// TwinCAT 3 PLC project PLC
// ProgramVersion: 3.1.4026.19
// CompilerDefines: VISU_USEPROPERTYINFO
// libraries:
//   SPT Base Types, * (Beckhoff Automation LLC)
//   SPT Components, * (Beckhoff Automation LLC)
//   SPT Motion Control, * (Beckhoff Automation LLC)
//   SPT Utilities, * (Beckhoff Automation LLC)
//   Tc2_Standard, * (Beckhoff Automation GmbH)
//   Tc2_System, * (Beckhoff Automation GmbH)
//   Tc3_PackML_V3, * (Beckhoff Automation GmbH)
// project tree:
//   DUTs/ E_PMLCustomMode.TcDUT, ST_ModeList.TcDUT
//   / GlobalTextList.TcGTLO, PlcTask.TcTTO, Visualization Manager.TcVMO (not stored)
//   Modes/ FB_CustomModes.TcPOU
//   Modules/00 Machine/DUTs/ ST_Machine_Command.TcDUT, ST_Machine_Config.TcDUT, ST_Machine_HMI.TcDUT, ST_Machine_Status.TcDUT
//   Modules/00 Machine/ Machine.TcPOU
//   Modules/01 Infeed/ Infeed.TcPOU
//   Modules/02 Process/ Process.TcPOU
//   Modules/03 Outfeed/ Outfeed.TcPOU
//   POUs/ MAIN.TcPOU
//   VISUs/ Visualization.TcVIS
// real-time tasks:
//   TASK PlcTask: cycle T#10ms, priority 20, ADS port 350
// motion (NC):
//   TASK NC-Task 1 SAF: cycle T#2ms, priority 4, ADS port 501
//   TASK NC-Task 1 SVB: cycle T#10ms, priority 8, ADS port 511
//   AXIS Axis 1 (id 1)
// variable links:
//   PLC/PLC Instance <-> NC-Task 1 SAF/Axes/Axis 1
//     PlcTask Inputs/MAIN.Machine.Infeed.Axis.BasicAxis._Axis.NcToPlc <-> Outputs/ToPlc
//     PlcTask Outputs/MAIN.Machine.Infeed.Axis.BasicAxis._Axis.PlcToNc <-> Inputs/FromPlc

CONFIGURATION PLC
    RESOURCE PLC ON TwinCAT3
        TASK PlcTask(INTERVAL := T#10ms, PRIORITY := 20);
        PROGRAM MAIN WITH PlcTask : MAIN;
    END_RESOURCE
END_CONFIGURATION

// ---- DUTs/E_PMLCustomMode.TcDUT
{attribute 'to_string'}
TYPE E_PMLCustomMode : (
		//Protected
		Invalid		:= 0,
		Production	:= 1,
		Maintenance := 2,
		Manual		:= 3,
		//User-Defined
		Home		  := 4,	 //User Mode 1
		PrePosition	  := 5,	 //User Mode 2
		PreProduction := 6,	 //User Mode 3
		SingleCycle	  := 7,	 //User Mode 4
		SingleStep	  := 8,	 //User Mode 5
		Setup		  := 9,	 //User Mode 6
		CleanInPlace  := 10, //User Mode 7
		DryCycle	  := 11, //User Mode 8
		Teach		  := 12, //User Mode 9
		Remote		  := 13, //User Mode 10
		Last		  := 14	 //User Mode 11

	//E_PMLUnitMode.ePMLUnitMode_UserMode28
	) DINT;
END_TYPE

// ---- DUTs/ST_ModeList.TcDUT
TYPE ST_ModeList :
	STRUCT
		// Protected
		Invalid		: BOOL;
		Production	: BOOL;
		Maintenance : BOOL;
		Manual		: BOOL;
		// User-Defined
		Home		  : BOOL;
		PrePosition	  : BOOL;
		PreProduction : BOOL;
		SingleCycle	  : BOOL;
		SingleStep	  : BOOL;
		Setup		  : BOOL;
		CleanInPlace  : BOOL;
		DryCycle	  : BOOL;
		Teach		  : BOOL;
		Remote		  : BOOL;
		Last		  : BOOL;
		// Unused
		UserMode12 : BOOL;
		UserMode13 : BOOL;
		UserMode14 : BOOL;
		UserMode15 : BOOL;
		UserMode16 : BOOL;
		UserMode17 : BOOL;
		UserMode18 : BOOL;
		UserMode19 : BOOL;
		UserMode20 : BOOL;
		UserMode21 : BOOL;
		UserMode22 : BOOL;
		UserMode23 : BOOL;
		UserMode24 : BOOL;
		UserMode25 : BOOL;
		UserMode26 : BOOL;
		UserMode27 : BOOL;
		UserMode28 : BOOL;
	END_STRUCT
END_TYPE

// ---- Modules/00 Machine/DUTs/ST_Machine_Command.TcDUT
TYPE ST_Machine_Command :
	STRUCT
		StartHoming : BOOL;
	END_STRUCT
END_TYPE

// ---- Modules/00 Machine/DUTs/ST_Machine_Config.TcDUT
TYPE ST_Machine_Config :
	STRUCT
	END_STRUCT
END_TYPE

// ---- Modules/00 Machine/DUTs/ST_Machine_HMI.TcDUT
TYPE ST_Machine_HMI :
	STRUCT
		Command : ST_Machine_Command;
		Config	: ST_Machine_Config;
		Status	: ST_Machine_Status;
	END_STRUCT
END_TYPE

// ---- Modules/00 Machine/DUTs/ST_Machine_Status.TcDUT
TYPE ST_Machine_Status :
	STRUCT
		HomeComplete  : BOOL;
		NeedsCleaning : BOOL;
		CleanComplete : BOOL;
	END_STRUCT
END_TYPE

// ---- POUs/MAIN.TcPOU
PROGRAM MAIN
VAR
	Machine : Machine := (Name := 'Machine');
END_VAR

(*All sample code provided by Beckhoff Automation LLC are for illustrative purposes only and are provided “as is” and without any warranties, express or implied. Actual implementations in applications will vary significantly. Beckhoff Automation LLC shall have no liability for, and does not waive any rights in relation to, any code samples that it provides or the use of such code samples for any purpose.*)

(*
	This sample demonstrates changing mode based on the status of the machine.
	Specifically on startup, the Machine Status for HomeComplete is FALSE.
	Therefore in Machine.Idle the mode is changed to Home.
	When the 'Start command is given the Machine can then Execute its Homing routine, Complete, and then return to Idle.
	Once back in Idle, the Machine status of HomeComplete will retunr the mode to Production.
*)
Machine.CyclicLogic();

END_PROGRAM

// ---- Modules/00 Machine/Machine.TcPOU
FUNCTION_BLOCK Machine EXTENDS FB_PackML_BaseModule
VAR
	Infeed	: Infeed  := (Name := 'Infeed');
	Process : Process := (Name := 'Process');
	Outfeed : Outfeed := (Name := 'Outfeed');

	//
	Machine_HMI		  : ST_Machine_HMI;
	CurrentCustomMode : E_PMLCustomMode;
END_VAR

METHOD CreateCustomModes
VAR
	i		   : E_PMLCustomMode;
	aModeNames : ARRAY[E_PMLCustomMode.Invalid..E_PMLCustomMode.Last] OF STRING;
END_VAR
aModeNames[0]  := TO_STRING(E_PMLCustomMode.Invalid);
aModeNames[1]  := TO_STRING(E_PMLCustomMode.Production);
aModeNames[2]  := TO_STRING(E_PMLCustomMode.Maintenance);
aModeNames[3]  := TO_STRING(E_PMLCustomMode.Manual);
aModeNames[4]  := TO_STRING(E_PMLCustomMode.Home);			//UserMode1
aModeNames[5]  := TO_STRING(E_PMLCustomMode.PrePosition);	//UserMode2
aModeNames[6]  := TO_STRING(E_PMLCustomMode.PreProduction); //UserMode3
aModeNames[7]  := TO_STRING(E_PMLCustomMode.SingleCycle);	//UserMode4
aModeNames[8]  := TO_STRING(E_PMLCustomMode.SingleStep);	//UserMode5
aModeNames[9]  := TO_STRING(E_PMLCustomMode.Setup);			//UserMode6
aModeNames[10] := TO_STRING(E_PMLCustomMode.CleanInPlace);	//UserMode7
aModeNames[11] := TO_STRING(E_PMLCustomMode.DryCycle);		//UserMode8
aModeNames[12] := TO_STRING(E_PMLCustomMode.Teach);			//UserMode9
aModeNames[13] := TO_STRING(E_PMLCustomMode.Remote);		//UserMode10
aModeNames[14] := TO_STRING(E_PMLCustomMode.Last);			//UserMode11

//Default Config for all modes, this is also the default config for Production Mode as defined by Pack ML
CustomModes.bDisableClearing			   := FALSE;
CustomModes.bDisableStarting			   := FALSE;
CustomModes.bDisableSuspended			   := FALSE;
CustomModes.bDisableStopping			   := FALSE;
CustomModes.bDisableAborting			   := FALSE;
CustomModes.bDisableHolding				   := FALSE;
CustomModes.bDisableHeld				   := FALSE;
CustomModes.bDisableUnholding			   := FALSE;
CustomModes.bDisableSuspending			   := FALSE;
CustomModes.bDisableUnsuspending		   := FALSE;
CustomModes.bDisableResetting			   := FALSE;
CustomModes.bDisableIdle				   := FALSE;
CustomModes.bDisableCompleting			   := FALSE;
CustomModes.bDisableComplete			   := FALSE;
CustomModes.bEnableUnitModeChangeStopped   := TRUE;
CustomModes.bEnableUnitModeChangeIdle	   := TRUE;
CustomModes.bEnableUnitModeChangeSuspended := TRUE;
CustomModes.bEnableUnitModeChangeExecute   := FALSE;
CustomModes.bEnableUnitModeChangeAborted   := TRUE;
CustomModes.bEnableUnitModeChangeHeld	   := TRUE;
CustomModes.bEnableUnitModeChangeComplete  := TRUE;

//
FOR i := E_PMLCustomMode.Invalid TO E_PMLCustomMode.Last DO
	CustomModes(emode := i, sName := aModeNames[i]);
END_FOR

// Production - Changes for Clean In Place Mode to move from Production.Execute to CleanInPlace.Execute
CustomModes(eMode := E_PMLCustomMode.Production, sName := 'Production', bEnableUnitModeChangeExecute := TRUE);

//Maintenance Mode default as defined by PackML
CustomModes(eMode						   := E_PMLCustomMode.Maintenance,
			sName						   := 'Maintenance',
			bDisableClearing			   := FALSE,
			bDisableStarting			   := FALSE,
			bDisableSuspended			   := TRUE,
			bDisableStopping			   := FALSE,
			bDisableAborting			   := FALSE,
			bDisableHolding				   := FALSE,
			bDisableHeld				   := FALSE,
			bDisableUnholding			   := FALSE,
			bDisableSuspending			   := TRUE,
			bDisableUnsuspending		   := TRUE,
			bDisableResetting			   := FALSE,
			bDisableIdle				   := FALSE,
			bDisableCompleting			   := TRUE,
			bDisableComplete			   := TRUE,
			bEnableUnitModeChangeStopped   := TRUE,
			bEnableUnitModeChangeIdle	   := TRUE,
			bEnableUnitModeChangeSuspended := FALSE,
			bEnableUnitModeChangeExecute   := FALSE,
			bEnableUnitModeChangeAborted   := TRUE,
			bEnableUnitModeChangeHeld	   := TRUE,
			bEnableUnitModeChangeComplete  := FALSE);

//Manual Mode default as defined by PackML
CustomModes(eMode						   := E_PMLCustomMode.Manual,
			sName						   := 'Manual',
			bDisableClearing			   := FALSE,
			bDisableStarting			   := FALSE,
			bDisableSuspended			   := TRUE,
			bDisableStopping			   := FALSE,
			bDisableAborting			   := FALSE,
			bDisableHolding				   := TRUE,
			bDisableHeld				   := TRUE,
			bDisableUnholding			   := TRUE,
			bDisableSuspending			   := TRUE,
			bDisableUnsuspending		   := TRUE,
			bDisableResetting			   := FALSE,
			bDisableIdle				   := FALSE,
			bDisableCompleting			   := TRUE,
			bDisableComplete			   := TRUE,
			bEnableUnitModeChangeStopped   := TRUE,
			bEnableUnitModeChangeIdle	   := TRUE,
			bEnableUnitModeChangeSuspended := FALSE,
			bEnableUnitModeChangeExecute   := FALSE,
			bEnableUnitModeChangeAborted   := TRUE,
			bEnableUnitModeChangeHeld	   := FALSE,
			bEnableUnitModeChangeComplete  := FALSE);

//Home Mode - Configured the same as Production as Defined by PackML
CustomModes(eMode						   := E_PMLCustomMode.Home,
			sName						   := 'Home',
			bDisableClearing			   := FALSE,
			bDisableStarting			   := FALSE,
			bDisableSuspended			   := FALSE,
			bDisableStopping			   := FALSE,
			bDisableAborting			   := FALSE,
			bDisableHolding				   := FALSE,
			bDisableHeld				   := FALSE,
			bDisableUnholding			   := FALSE,
			bDisableSuspending			   := FALSE,
			bDisableUnsuspending		   := FALSE,
			bDisableResetting			   := FALSE,
			bDisableIdle				   := FALSE,
			bDisableCompleting			   := FALSE,
			bDisableComplete			   := FALSE,
			bEnableUnitModeChangeStopped   := TRUE,
			bEnableUnitModeChangeIdle	   := TRUE,
			bEnableUnitModeChangeSuspended := TRUE,
			bEnableUnitModeChangeExecute   := FALSE,
			bEnableUnitModeChangeAborted   := TRUE,
			bEnableUnitModeChangeHeld	   := TRUE,
			bEnableUnitModeChangeComplete  := TRUE);

// Dry Cycle - If settings are the same as Production, only the eMode and sName must be updated
CustomModes(eMode := E_PMLCustomMode.DryCycle, sName := 'Dry Cycle');

// Teach - If settings are similar to Production, only the eMode, sName, and the differences must be changed
CustomModes(eMode						   := E_PMLCustomMode.Teach,
			sName						   := 'Teach',
			bDisableHolding				   := TRUE,
			bDisableSuspending			   := TRUE,
			bEnableUnitModeChangeSuspended := FALSE,
			bEnableUnitModeChangeHeld	   := FALSE,
			bEnableUnitModeChangeComplete  := FALSE);

//This mode is not intended to be used
CustomModes(eMode						   := E_PMLCustomMode.Last,
			sName						   := 'Last',
			bDisableClearing			   := TRUE,
			bDisableStarting			   := TRUE,
			bDisableSuspended			   := TRUE,
			bDisableStopping			   := TRUE,
			bDisableAborting			   := FALSE,
			bDisableHolding				   := TRUE,
			bDisableHeld				   := TRUE,
			bDisableUnholding			   := TRUE,
			bDisableSuspending			   := TRUE,
			bDisableUnsuspending		   := TRUE,
			bDisableResetting			   := TRUE,
			bDisableIdle				   := TRUE,
			bDisableCompleting			   := TRUE,
			bDisableComplete			   := TRUE,
			bEnableUnitModeChangeStopped   := FALSE,
			bEnableUnitModeChangeIdle	   := FALSE,
			bEnableUnitModeChangeSuspended := FALSE,
			bEnableUnitModeChangeExecute   := FALSE,
			bEnableUnitModeChangeAborted   := TRUE,
			bEnableUnitModeChangeHeld	   := FALSE,
			bEnableUnitModeChangeComplete  := FALSE);

//Clean In Place - 
CustomModes(eMode						   := E_PMLCustomMode.CleanInPlace,
			sName						   := 'Clean In Place',
			bDisableClearing			   := FALSE,
			bDisableStarting			   := FALSE,
			bDisableSuspended			   := FALSE,
			bDisableStopping			   := FALSE,
			bDisableAborting			   := FALSE,
			bDisableHolding				   := TRUE,
			bDisableHeld				   := TRUE,
			bDisableUnholding			   := TRUE,
			bDisableSuspending			   := TRUE,
			bDisableUnsuspending		   := TRUE,
			bDisableResetting			   := FALSE,
			bDisableIdle				   := FALSE,
			bDisableCompleting			   := FALSE,
			bDisableComplete			   := FALSE,
			bEnableUnitModeChangeStopped   := TRUE,
			bEnableUnitModeChangeIdle	   := TRUE,
			bEnableUnitModeChangeSuspended := FALSE,
			bEnableUnitModeChangeExecute   := TRUE,
			bEnableUnitModeChangeAborted   := TRUE,
			bEnableUnitModeChangeHeld	   := FALSE,
			bEnableUnitModeChangeComplete  := FALSE);
END_METHOD

METHOD CyclicLogic
VAR
END_VAR
IF NOT _InitComplete THEN
	_InitComplete := Initialize();
	RETURN;
END_IF

CurrentCustomMode := _CurrentMode;

//
SUPER^.CyclicLogic();
END_METHOD

(* This method contains code which will execute when this PackML module is in the Execute state*)
METHOD PROTECTED Execute
VAR
END_VAR
CASE _CurrentMode OF
	E_PMLCustomMode.Production:
		IF Machine_HMI.Status.NeedsCleaning THEN
			ChangeMode(Mode := E_PMLCustomMode.CleanInPlace);
		END_IF

	E_PMLCustomMode.Home: //User Mode 1
		IF Machine_HMI.Command.StartHoming THEN
			Machine_HMI.Command.StartHoming := FALSE;
			Machine_HMI.Status.HomeComplete := TRUE;
			ChangeState(State := E_PMLCommand.Complete);
		END_IF

	E_PMLCustomMode.SingleCycle:
	E_PMLCustomMode.Maintenance:
		;

	E_PMLCustomMode.CleanInPlace:
		IF Machine_HMI.Status.CleanComplete THEN
			ChangeMode(Mode := E_PMLCustomMode.Production);
		END_IF

ELSE
	;
END_CASE
END_METHOD

(* Automatically enables and disables HMI control based on the PackML mode*)
METHOD PROTECTED HMIPermissions
AllowHMIControl(TRUE);
END_METHOD

(* This method contains code which will execute when this PackML module is in the Idle state*)
METHOD PROTECTED Idle
CASE _CurrentMode OF
	E_PMLCustomMode.Production:
		IF NOT Machine_HMI.Status.HomeComplete THEN
			ChangeMode(Mode := E_PMLCustomMode.Home);
		END_IF

	E_PMLCustomMode.Home: //User Mode 1
		IF Machine_HMI.Status.HomeComplete THEN
			ChangeMode(Mode := E_PMLCustomMode.Production);
		END_IF

	E_PMLCustomMode.Maintenance:
		;

	E_PMLCustomMode.Manual:
		;

ELSE // Current Mode not accounted for
	Trace(Message := CONCAT(TO_STRING(_CurrentMode), ' not handled in state Idle'));
	ChangeState(State := E_PMLCommand.Abort);
END_CASE
END_METHOD

(* Basic module initialization logic*)
METHOD PROTECTED Initialize : BOOL
Initialize := FALSE;
CASE DescendantSequenceState OF
	0:
		RegisterSubmodule(SubModule := Infeed);
		RegisterSubmodule(SubModule := Process);
		RegisterSubmodule(SubModule := Outfeed);
		DescendantSequenceState := DescendantSequenceState + 10;

	10:
		CreateCustomModes();
		DescendantSequenceState := DescendantSequenceState + 10;

	20:
		IF SUPER^.Initialize() THEN
			DescendantSequenceState := DescendantSequenceState + 10;
		END_IF

	30:
		Initialize := TRUE;
END_CASE
END_METHOD

END_FUNCTION_BLOCK

// ---- Modules/01 Infeed/Infeed.TcPOU
FUNCTION_BLOCK Infeed EXTENDS FB_PackML_BaseModule
VAR
	Axis			  : FB_Component_BasicAxis;
	CurrentCustomMode : E_PMLCustomMode;
	_Start			  : BOOL;
	_Stop			  : BOOL;
END_VAR

METHOD CyclicLogic
IF NOT _InitComplete THEN
	_InitComplete := Initialize();
	RETURN;
END_IF

CurrentCustomMode := _CurrentMode;

//
SUPER^.CyclicLogic();
END_METHOD

(* This method contains code which will execute when this PackML module is in the Execute state*)
METHOD PROTECTED Execute
VAR
END_VAR
CASE _CurrentMode OF
	E_PMLCustomMode.Manual:
		IF _Stop THEN
			_Stop := FALSE;
			ChangeState(State := E_PMLCommand.Stop);
		END_IF

	E_PMLCustomMode.Production:

	//Waiting for Machine
END_CASE
END_METHOD

(* This method contains code which will execute when this PackML module is in the Idle state*)
METHOD PROTECTED Idle
VAR
END_VAR
CASE _CurrentMode OF
	E_PMLCustomMode.Manual:
		IF _Start THEN
			_Start := FALSE;
			ChangeState(State := E_PMLCommand.Start);
		END_IF

	E_PMLCustomMode.Production:

	//Waiting for Machine
END_CASE
END_METHOD

(* Basic module initialization logic*)
METHOD PROTECTED Initialize : BOOL
CASE DescendantSequenceState OF
	0:
		RegisterComponent(Axis);
		DescendantSequenceState := DescendantSequenceState + 10;

	10:
		IF SUPER^.Initialize() THEN
			Initialize := TRUE;
		END_IF
END_CASE
END_METHOD

END_FUNCTION_BLOCK

// ---- Modules/02 Process/Process.TcPOU
FUNCTION_BLOCK Process EXTENDS FB_PackML_BaseModule
VAR
	CurrentCustomMode : E_PMLCustomMode;
END_VAR

METHOD CyclicLogic
VAR
	_Start : BOOL;
END_VAR
IF NOT _InitComplete THEN
	_InitComplete := Initialize();
	RETURN;
END_IF

CurrentCustomMode := _CurrentMode;

//
SUPER^.CyclicLogic();
END_METHOD

END_FUNCTION_BLOCK

// ---- Modules/03 Outfeed/Outfeed.TcPOU
FUNCTION_BLOCK Outfeed EXTENDS FB_PackML_BaseModule
VAR
	CurrentCustomMode : E_PMLCustomMode;
END_VAR

METHOD CyclicLogic
IF NOT _InitComplete THEN
	_InitComplete := Initialize();
	RETURN;
END_IF

CurrentCustomMode := _CurrentMode;

//
SUPER^.CyclicLogic();
END_METHOD

END_FUNCTION_BLOCK

// ---- Modes/FB_CustomModes.TcPOU
FUNCTION_BLOCK FB_CustomModes EXTENDS FB_CyclicFB IMPLEMENTS I_ModeList
VAR
	ModeList : ST_ModeList;
	ipModes	 : I_ModeList;
END_VAR

METHOD CyclicLogic
END_METHOD

//FB_Init is always available implicitly and it is used primarily for initialization.

//The return value is not evaluated. For a specific influence, you can also declare the

//methods explicitly and provide additional code there with the standard initialization

//code. You can evaluate the return value.
METHOD FB_Init : BOOL
VAR_INPUT
	bInitRetains : BOOL; // TRUE: the retain variables are initialized (reset warm / reset cold)
	bInCopyCode	 : BOOL; // TRUE: the instance will be copied to the copy code afterward (online change)   
END_VAR
ModeList := ModeNames;
END_METHOD

PROPERTY ModeNames : REFERENCE TO ST_ModeList
GET
ModeNames REF= ipModes.ModeNames;
END_GET
SET
ModeList := ModeNames;
END_SET
END_PROPERTY

END_FUNCTION_BLOCK

// ---- GlobalTextList.TcGTLO
TEXTLIST GlobalTextList
  792 = '%s'
  834 = 'Current Mode: %s'
  275 = 'Home Command'
  976 = 'Home Status'
  997 = 'Next Available Commnds'
  686 = 'Next Available State Commnds'
END_TEXTLIST

// ---- VISUs/Visualization.TcVIS
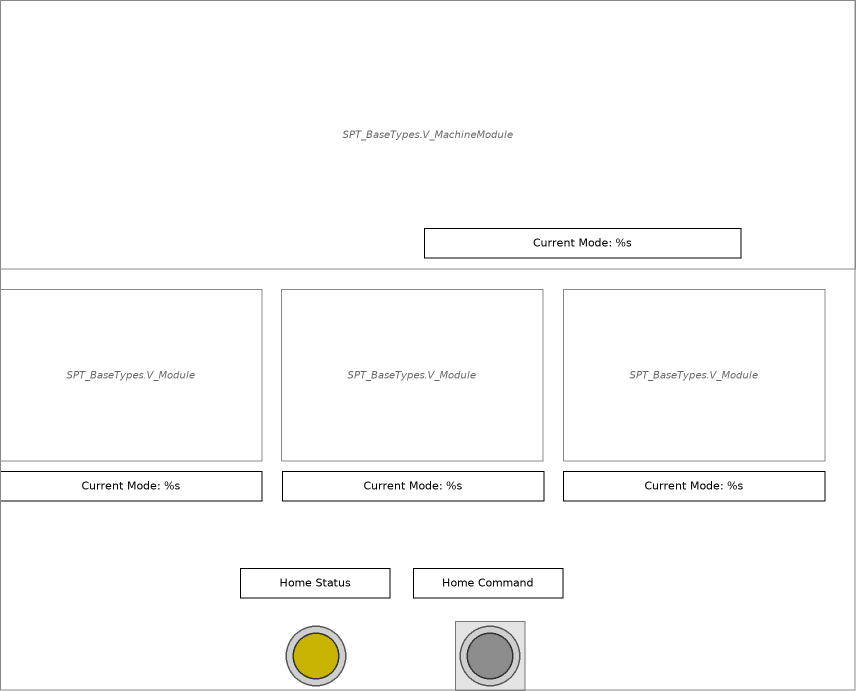
VISUALIZATION Visualization  // 856x691
    Frame (0,0 856x269)
        shows SPT_BaseTypes.V_MachineModule(HMI := MAIN.Machine.PackMLBaseModule_HMI)
    Lamp1 (281,621 70x70), variable: MAIN.Machine.Machine_HMI.Status.HomeComplete, style: Lamp-Lamp1-Yellow
    PushSwitch (455,621 70x70), variable: MAIN.Machine.Machine_HMI.Command.StartHoming, behaviour: TOGGLE, style: Switch-PushSwitch-Gray
    Rectangle (240,568 150x30), "Home Status"
    Rectangle (413,568 150x30), "Home Command"
    Frame (0,289 262x172)
        shows SPT_BaseTypes.V_Module(HMI := MAIN.Machine.Infeed.PackMLBaseModule_HMI)
    Frame (281,289 262x172)
        shows SPT_BaseTypes.V_Module(HMI := MAIN.Machine.Process.PackMLBaseModule_HMI)
    Frame (563,289 262x172)
        shows SPT_BaseTypes.V_Module(HMI := MAIN.Machine.Outfeed.PackMLBaseModule_HMI)
    Rectangle (424,228 317x30), "Current Mode: %s", text variable: MAIN.Machine.CurrentCustomMode
    Rectangle (0,471 262x30), "Current Mode: %s", text variable: MAIN.Machine.Infeed.CurrentCustomMode
    Rectangle (282,471 262x30), "Current Mode: %s", text variable: MAIN.Machine.Process.CurrentCustomMode
    Rectangle (563,471 262x30), "Current Mode: %s", text variable: MAIN.Machine.Outfeed.CurrentCustomMode
END_VISUALIZATION
